INTERFACE ITF_BaseTime

END_INTERFACE

(* stored: Version 1.1.0.1
   Itf ITF_BaseTime: Id {b1a3bb1d-6bec-0fd1-09bc-0dce04dcea5e} *)
